Fanuc KAREL source: compact_preamble.KL

PROGRAM KX00021
%NOLOCKGROUP
VAR
I:INTEGER;J:INTEGER;B:BOOLEAN
F : FILE
S : STRING[80]
P : XYZWPR
AA : ARRAY[2,3] OF INTEGER
BEGIN
AA[1,2]=4
I=AA[1,2]
END KX00021
